Universal Robots URScript: 27- force_simple.script

def P27_force_simple():
  set_standard_analog_input_domain(0, 1)
  set_standard_analog_input_domain(1, 1)
  set_tool_analog_input_domain(0, 1)
  set_tool_analog_input_domain(1, 1)
  set_analog_outputdomain(0, 0)
  set_analog_outputdomain(1, 0)
  set_tool_voltage(0)
  set_tcp(p[0.0,0.0,0.0,0.0,0.0,0.0])
  set_payload(0.0)
  set_gravity([0.0, 0.0, 9.82])
  global i_var_1=0
  while (True):
    $ 1 "机器人程序"
    $ 2 "MoveL"
    $ 3 "路点_1"
    movel([-0.7131688962876446, -1.6173202298344123, -1.536981164405514, -1.5554655565397457, 1.6060771732863524, 0.8568899973333854], a=1.2, v=0.25)
    $ 4 "路点_2"
    movel([-0.7131688964017702, -1.8723134037429974, -2.0238798389059083, -0.8135737081348609, 1.6060771732866534, 0.8568899972192523], a=1.2, v=0.25)
    sync()
    force_mode(p[0.0,0.0,0.0,0.0,0.0,0.0], [0, 0, 1, 0, 0, 0], [0.0, 0.0, 20.0, 0.0, 0.0, 0.0], 2, [0.1, 0.1, 0.15, 0.3490658503988659, 0.3490658503988659, 0.3490658503988659])
    $ 5 "力"
    $ 6 "路点_2"
    movel([-0.7131688964017702, -1.8723134037429974, -2.0238798389059083, -0.8135737081348609, 1.6060771732866534, 0.8568899972192523], a=1.2, v=0.25)
    $ 7 "路点_3"
    movel([0.38834304082772153, -1.3994211895149, -2.5535697890579687, -0.7267438884027353, 1.5844120173812535, 1.958578003636596], a=1.2, v=0.25)
    end_force_mode()
    stopl(5.0)
    $ 8 "路点_4"
    movel([0.38834304103178585, -1.1021315610482878, -1.9220721976165098, -1.6555311083080282, 1.5844120173747958, 1.9585780038406497], a=1.2, v=0.25)
  end
end
